(* IEC 61131-3 sources: AXOpen/src/components.siem.identification/ctrl/src/AxoSimaticIdentCyclic/TypesStructuresAndEnums, 9 files *)

(* ---- eAxoSimaticIdentCyclic_IOsize.st ---- *)
NAMESPACE AXOpen.Components.Siem.Identification
   TYPE PUBLIC
      eAxoSimaticIdentCyclic_IOsize : UINT
       (
         INVALID     := UINT#0,
         BYTES_32    := UINT#32,
         BYTES_116   := UINT#116,
         BYTES_128   := UINT#128
         );
   END_TYPE
END_NAMESPACE

(* ---- eAxoSimaticIdentCyclic_Port.st ---- *)
NAMESPACE AXOpen.Components.Siem.Identification
   TYPE PUBLIC
       eAxoSimaticIdentCyclic_Port : UINT
       (
         NONE  := UINT#0,
         X21   := UINT#2,
         X22   := UINT#3
         );
   END_TYPE
END_NAMESPACE

(* ---- AxoSimaticIdentCyclic_Component_Status.st ---- *)
NAMESPACE AXOpen.Components.Siem.Identification
    {S7.extern=ReadWrite}
    {#ix-attr:[Container(Layout.Stack)]}
    CLASS PUBLIC AxoSimaticIdentCyclic_Component_Status EXTENDS AXOpen.Components.Abstractions.AxoComponent_Status
        VAR PUBLIC

        END_VAR
    END_CLASS
END_NAMESPACE

(* ---- AxoSimaticIdentCyclic_Config.st ---- *)
NAMESPACE AXOpen.Components.Siem.Identification
    {S7.extern=ReadWrite}
    {#ix-attr:[Container(Layout.Stack)]}
    CLASS PUBLIC AxoSimaticIdentCyclic_Config
        VAR PUBLIC
            {#ix-set:AttributeName = "<#Info time#>"}
            InfoTime : LTIME := LT#5S;
            {#ix-set:AttributeName = "<#Error time#>"}
            ErrorTime : LTIME := LT#10S;
            {#ix-set:AttributeName = "<#Port#>"}
            Port    : eAxoSimaticIdentCyclic_Port := eAxoSimaticIdentCyclic_Port#NONE;
            {#ix-set:AttributeName = "<#Reader IO image size (in bytes)#>"}
            IOsize  : eAxoSimaticIdentCyclic_IOsize := eAxoSimaticIdentCyclic_IOsize#INVALID;
            {#ix-set:AttributeName = "<#Hardware IDs#>"}
            HWIDs : AxoSimaticIdentCyclic_HWIDs;
            {#ix-set:AttributeName = "<#Data buffer low index#>"}
            DataBufferLowIndex  :  INT;
            {#ix-set:AttributeName = "<#Data buffer high index#>"}
            DataBufferHighIndex :  INT;
        END_VAR
    END_CLASS
END_NAMESPACE

(* ---- AxoSimaticIdentCyclic_Control.st ---- *)
NAMESPACE AXOpen.Components.Siem.Identification
    {S7.extern=ReadWrite}
    {#ix-attr:[Container(Layout.Stack)]}
    CLASS PUBLIC AxoSimaticIdentCyclic_Control
        VAR PUBLIC
            {#ix-set:AttributeName = "<#Start#>"}
            START 			:	BOOL;
            {#ix-set:AttributeName = "<#Reset#>"}
            RESET 			:	BOOL;
            {#ix-set:AttributeName = "<#Stop#>"}
            STOP 			:	BOOL;
            {#ix-set:AttributeName = "<#Switch off antenna#>"}
            ANTOFF 			:	BOOL;
            {#ix-set:AttributeName = "<#Block#>"}
            BLOCK 			    :	BOOL;
            {#ix-set:AttributeName = "<#Command#>"}
            CMD 			    :	BOOL;
            {#ix-set:AttributeName = "<#Index of the tag field#>"}
            TAGFIELD            :   WORD;
            {#ix-set:AttributeName = "<#Start address on the transponder#>"}
            ADDRESS             :   DWORD;
            {#ix-set:AttributeName = "<#Length of the data#>"}
            LENGTH              :   WORD;
        END_VAR
    END_CLASS
END_NAMESPACE

(* ---- AxoSimaticIdentCyclic_HWIDs.st ---- *)
NAMESPACE AXOpen.Components.Siem.Identification
   {S7.extern=ReadWrite}
	CLASS AxoSimaticIdentCyclic_HWIDs
      VAR PUBLIC
         {#ix-set:AttributeName = "<#Hardware ID 'Head' submodule#>"}
         HW_Head              :  UINT;
         {#ix-set:AttributeName = "<#Hardware ID 'CM' submodule#>"}
         HwID_CM              :   UINT;
         {#ix-set:AttributeName = "<#Hardware ID 'Reader' submodule#>"}
         HwID_Reader          :   UINT;
      END_VAR
   END_CLASS
END_NAMESPACE

(* ---- AxoSimaticIdentCyclic_In.st ---- *)
NAMESPACE AXOpen.Components.Siem.Identification
    {S7.extern=ReadWrite}
    {#ix-attr:[Container(Layout.Wrap)]}
    CLASS PUBLIC AxoSimaticIdentCyclic_In
        VAR PUBLIC
            {#ix-set:AttributeName = "<#Status#>"}
            {#ix-attr:[ReadOnly()]}
            Status  :   AxoSimaticIdentCyclic_Status;
            {#ix-attr:[ReadOnly()]}
            // {#ix-set:AttributeName = "<#Data#>"}
            Data    :   ARRAY[0..123] OF BYTE;
        END_VAR
    END_CLASS
END_NAMESPACE

(* ---- AxoSimaticIdentCyclic_Out.st ---- *)
NAMESPACE AXOpen.Components.Siem.Identification
    {S7.extern=ReadWrite}
    {#ix-attr:[Container(Layout.Wrap)]}
    CLASS PUBLIC AxoSimaticIdentCyclic_Out
        VAR PUBLIC
            {#ix-set:AttributeName = "<#Control#>"}
            {#ix-attr:[ReadOnly()]}
            Control           :   AxoSimaticIdentCyclic_Control;
            {#ix-set:AttributeName = "<#User data#>"}
            USER_DATA           :   ARRAY[0..123] OF BYTE;
        END_VAR
    END_CLASS
END_NAMESPACE

(* ---- AxoSimaticIdentCyclic_Status.st ---- *)
NAMESPACE AXOpen.Components.Siem.Identification
    {S7.extern=ReadWrite}
    {#ix-attr:[Container(Layout.Stack)]}
    CLASS PUBLIC AxoSimaticIdentCyclic_Status
        VAR PUBLIC

        END_VAR
    END_CLASS
END_NAMESPACE
